TYPE ST_LoadExperimentSetting :
STRUCT
	Weight : INT; 
	Test_Finished : BOOL; 
END_STRUCT
END_TYPE

(* stored: Version 1.1.0.1, ProductVersion 3.1.4024.12
   DUT ST_LoadExperimentSetting: Id {841fd751-6090-403f-bf49-45ef31826432} *)
